// TIA Portal V20 export
TYPE "typeEnMeterOutputData"
TITLE = Energy Meter Ausgangsdaten / Energy meter output data
// Struktur Energy Meter Ausgaenge / Structure energy meter output
// stored: Access Published
   STRUCT
      byte0 : Byte;   // Steuerbyte 0 / Control byte 0
      byte1Bit0 : Bool;   // Steuerbyte 1.0 / Control byte 1.0
      byte1Bit1 : Bool;   // Steuerbyte 1.1 / Control byte 1.1
      byte1Bit2 : Bool;   // Steuerbyte 1.2 / Control byte 1.2
      byte1Bit3 : Bool;   // Steuerbyte 1.3 / Control byte 1.3
      byte1Bit4 : Bool;   // Steuerbyte 1.4 / Control byte 1.4
      byte1Bit5 : Bool;   // Steuerbyte 1.5 / Control byte 1.5
      byte1Bit6 : Bool;   // Steuerbyte 1.6 / Control byte 1.6
      resetEnergyCounters : Bool;   // Reset alle Energie Zähler / Reset for energy counters
      byte2Bit0 : Bool;   // Steuerbyte 2.0 / Control byte 2.0
      byte2Bit1 : Bool;   // Steuerbyte 2.1 / Control byte 2.1
      byte2Bit2 : Bool;   // Steuerbyte 2.2 / Control byte 2.2
      byte2Bit3 : Bool;   // Steuerbyte 2.3 / Control byte 2.3
      byte2Bit4 : Bool;   // Steuerbyte 2.4 / Control byte 2.4
      resetActiveEnergy : Bool;   // Wirkenergie / Active Energy
      resetReactiveEnergy : Bool;   // Blindenergie / Reactive Energy
      resetApparentEnergy : Bool;   // Scheinenergie / Apparent Energy
      byte3 : Byte;   // Steuerbyte 3 / Control byte 3
      byte4 : Byte;   // Steuerbyte 4 / Control byte 4
      byte5 : Byte;   // Steuerbyte 5 / Control byte 5
      byte6 : Byte;   // Steuerbyte 6 / Control byte 6
      byte7 : Byte;   // Steuerbyte 7 / Control byte 7
      byte8 : Byte;   // Steuerbyte 8 / Control byte 8
      byte9 : Byte;   // Steuerbyte 9 / Control byte 9
      byte10 : Byte;   // Steuerbyte 10 / Control byte 10
      byte11 : Byte;   // Steuerbyte 11 / Control byte 11
   END_STRUCT;
END_TYPE
